// TIA Portal V18 export
DATA_BLOCK "idbControlSécheur"   // DB6
// stored: InstanceOfName nsSécheur.fbControlSécheur, InstanceOfType FB, Namespace nsSécheur
"nsSécheur.fbControlSécheur"
   // VAR_INPUT
   //    iIncreaseTemperature : Bool;
   //    iDecreaseTemperature : Bool;
   // END_VAR
   // VAR_IN_OUT
   //    ioTemperature : UInt;
   // END_VAR
BEGIN
END_DATA_BLOCK
